FUNCTION_BLOCK E_CTU (* Event-Driven Up Counter *)
  (* Standard: 61499-1-A.18; Classification: Event-driven blocks; Function: Up-counter *)
  (* Version 0.3, 2012-12-20, IH, TU Wien, added service sequences for test case specification *)
  (* Version 0.2, 2006-09-07, JHC, Holobloc Inc, Changed package to fb.rt.events. *)
  (* Version 0.1, 2001-04-27, JHC, Rockwell Automation, XML version *)
  (* Version 0.0, 1999-01-22, JHC, Rockwell Automation, SRC version *)
  (* Compiler header: package fb.rt.events; *)
  (* Compiler Java Sun JDK 1.5.0 *)
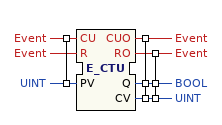
  EVENT_INPUT
    CU WITH PV; (* Count Up *)
    R; (* Reset *)
  END_EVENT
  EVENT_OUTPUT
    CUO WITH Q, CV; (* Count Up Output Event *)
    RO WITH Q, CV; (* Reset Output Event *)
  END_EVENT
  VAR_INPUT
    PV : UINT; (* Preset Value *)
  END_VAR
  VAR_OUTPUT
    Q : BOOL; (* CV>=PV *)
    CV : UINT;
  END_VAR
  SERVICE FB interface/Runtime Environment (* Event-Driven Up Counter *)
    SEQUENCE Initial Count-up
      FB interface.CU(PV:=5;) -> FB interface.CUO(Q:=FALSE;CV:=1;);
      FB interface.CU(PV:=5;) -> FB interface.CUO(Q:=FALSE;CV:=2;);
      FB interface.CU(PV:=5;) -> FB interface.CUO(Q:=FALSE;CV:=3;);
      FB interface.CU(PV:=5;) -> FB interface.CUO(Q:=FALSE;CV:=4;);
      FB interface.CU(PV:=5;) -> FB interface.CUO(Q:=TRUE;CV:=5;);
      FB interface.CU(PV:=5;) -> FB interface.CUO(Q:=TRUE;CV:=6;);
    END_SEQUENCE
    SEQUENCE Count up and reset with PV=0
      FB interface.R() -> FB interface.RO(Q:=FALSE;CV:=0;);
      FB interface.CU(PV:=0;) -> FB interface.CUO(Q:=TRUE;CV:=1;);
      FB interface.R() -> FB interface.RO(Q:=TRUE;CV:=0;);
      FB interface.CU(PV:=1;) -> FB interface.CUO(Q:=TRUE;CV:=1;);
    END_SEQUENCE
    SEQUENCE Count up with changing PV-values
      FB interface.R() -> FB interface.RO(Q:=FALSE;CV:=0;);
      FB interface.CU(PV:=1;) -> FB interface.CUO(Q:=TRUE;CV:=1;);
      FB interface.CU(PV:=3;) -> FB interface.CUO(Q:=FALSE;CV:=2;);
      FB interface.CU(PV:=3;) -> FB interface.CUO(Q:=TRUE;CV:=3;);
      FB interface.R() -> FB interface.RO(Q:=FALSE;CV:=0;);
    END_SEQUENCE
  END_SERVICE
END_FUNCTION_BLOCK
